Yaskawa INFORM job: P_X.JBI

/JOB
//NAME P_X
///FOLDERNAME INNE
//POS
///NPOS 7,7,7,0,0,0
///TOOL 0
///POSTYPE PULSE
///PULSE
C00000=75,7753,55829,25810,60260,35184
C00001=4674,8439,56820,49055,64050,31779
C00002=14033,-18,40155,76853,70936,31377
C00003=16176,-2606,31446,83912,74129,34922
C00004=-9786,3576,47748,174206,-59957,-42139
C00005=-13213,-856,38784,152241,-62450,-39168
C00006=-16589,-8630,22393,124282,-68179,-36921
BC00000=103636,1063120,678631
BC00001=103636,1063121,678632
BC00002=103636,1063121,678632
BC00003=103636,1063121,678632
BC00004=103636,1063121,678632
BC00005=103636,1063121,678632
BC00006=103636,1063121,678632
EC00000=1,1
EC00001=-167491,0
EC00002=-431280,0
EC00003=-525386,0
EC00004=274969,0
EC00005=440232,0
EC00006=678625,0
//INST
///DATE 2023/10/04 15:13
///ATTR SC,RW
///GROUP1 RB1,BS1
///GROUP2 ST1
NOP
MOVJ C00000 BC00000 VJ=0.78  +MOVJ EC00000 VJ=0.78
MOVJ C00001 BC00001 VJ=0.78  +MOVJ EC00001 VJ=0.78
MOVJ C00002 BC00002 VJ=0.78  +MOVJ EC00002 VJ=0.78
MOVJ C00003 BC00003 VJ=0.78  +MOVJ EC00003 VJ=0.78
MOVJ C00004 BC00004 VJ=0.78  +MOVJ EC00004 VJ=0.78
MOVJ C00005 BC00005 VJ=0.78  +MOVJ EC00005 VJ=0.78
MOVJ C00006 BC00006 VJ=0.78  +MOVJ EC00006 VJ=0.78
END
